// TIA Portal V18 export
DATA_BLOCK "ST10_DBInterface_Stopper"   // DB2602
{ S7_Optimized_Access := 'FALSE' }
VERSION : 0.1
// stored: AutoNumber false, DBAccessibleFromOPCUA true, DBAccessibleFromWebserver true, IsOnlyStoredInLoadMemory false, IsWriteProtectedInAS false
   VAR
      Stopper { S7_SetPoint := 'True'} : Array[1..50] of "UDT_StopperInterface";
   END_VAR
BEGIN
END_DATA_BLOCK
